LIN {X 0,Y 304.407,Z 934.466,A -85,B 0,C 180,E1 1225.073,E2 1225.073} C_VEL
LIN {X 0,Y 305.323,Z 932.612,A -85,B 0,C 180,E1 1225.322,E2 1225.322} C_VEL
LIN {X 0,Y 310.241,Z 921.537,A -85,B 0,C 180,E1 1225.913,E2 1225.913} C_VEL
LIN {X 0,Y 315.284,Z 909.54,A -85,B 0,C 180,E1 1226.349,E2 1226.349} C_VEL
LIN {X 0,Y 318.01,Z 902.452,A -85,B 0,C 180,E1 1226.415,E2 1226.415} C_VEL
LIN {X 0,Y 328.668,Z 871.537,A -85,B 0,C 180,E1 1226.315,E2 1226.315} C_VEL
LIN {X 0,Y 334.259,Z 852.306,A -85,B 0,C 180,E1 1226.308,E2 1226.308} C_VEL
LIN {X 0,Y 334.378,Z 852.639,A -85,B 0,C 180,E1 1227.359,E2 1227.359} C_VEL
LIN {X 0,Y 325.243,Z 882.784,A -85,B 0,C 180,E1 1227.209,E2 1227.209} C_VEL
LIN {X 0,Y 316.664,Z 906.295,A -85,B 0,C 180,E1 1226.963,E2 1226.963} C_VEL
LIN {X 0,Y 306.601,Z 930.253,A -85,B 0,C 180,E1 1226.554,E2 1226.554} C_VEL
LIN {X 0,Y 316.992,Z 905.088,A -85,B 0,C 180,E1 1226.427,E2 1226.427} C_VEL
LIN {X 0,Y 318.01,Z 902.452,A -85,B 0,C 180,E1 1226.415,E2 1226.415} C_VEL
LIN {X 0,Y 321.868,Z 903.174,A -85,B 0,C 180,E1 1226.375,E2 1226.375} C_VEL
LIN {X 0,Y 321.868,Z 1292,A -85,B 0,C 180,E1 1226.375,E2 1226.375} C_VEL
LIN {X 0,Y 321.868,Z 1292,A -85,B 0,C 180,E1 1226.375,E2 1226.375}

QRS_NEXT_CUT()

QRS_NEXT()
QRS_HOME()

END
